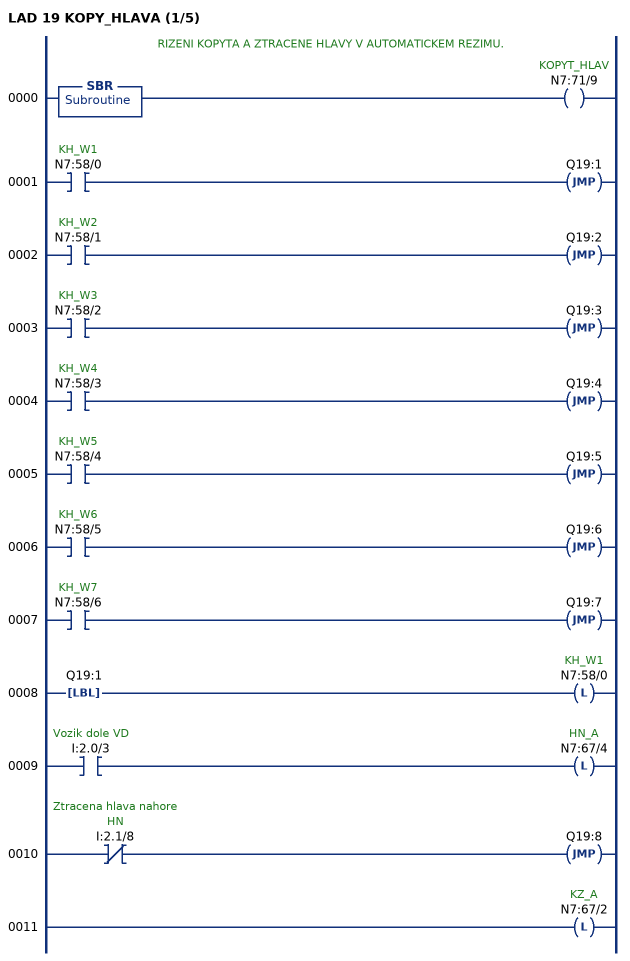
% Rung: 0 %
% RIZENI KOPYTA A ZTRACENE HLAVY V AUTOMATICKEM REZIMU. %
SOR SBR OTE N7:71/9 EOR
%   N7:71/9  KOPYT_HLAV %
% Rung: 1 %
SOR XIC N7:58/0 JMP Q19:1 EOR
%   N7:58/0  KH_W1 %
% Rung: 2 %
SOR XIC N7:58/1 JMP Q19:2 EOR
%   N7:58/1  KH_W2 %
% Rung: 3 %
SOR XIC N7:58/2 JMP Q19:3 EOR
%   N7:58/2  KH_W3 %
% Rung: 4 %
SOR XIC N7:58/3 JMP Q19:4 EOR
%   N7:58/3  KH_W4 %
% Rung: 5 %
SOR XIC N7:58/4 JMP Q19:5 EOR
%   N7:58/4  KH_W5 %
% Rung: 6 %
SOR XIC N7:58/5 JMP Q19:6 EOR
%   N7:58/5  KH_W6 %
% Rung: 7 %
SOR XIC N7:58/6 JMP Q19:7 EOR
%   N7:58/6  KH_W7 %
% Rung: 8 %
SOR LBL Q19:1 OTL N7:58/0 EOR
%   N7:58/0  KH_W1 %
% Rung: 9 %
SOR XIC I:2.0/3 OTL N7:67/4 EOR
%   I:2.0/3  VD  "Vozik dole" %
%   N7:67/4  HN_A %
% Rung: 10 %
SOR XIO I:2.1/8 JMP Q19:8 EOR
%   I:2.1/8  HN  "Ztracena hlava nahore" %
% Rung: 11 %
SOR OTL N7:67/2 EOR
%   N7:67/2  KZ_A %

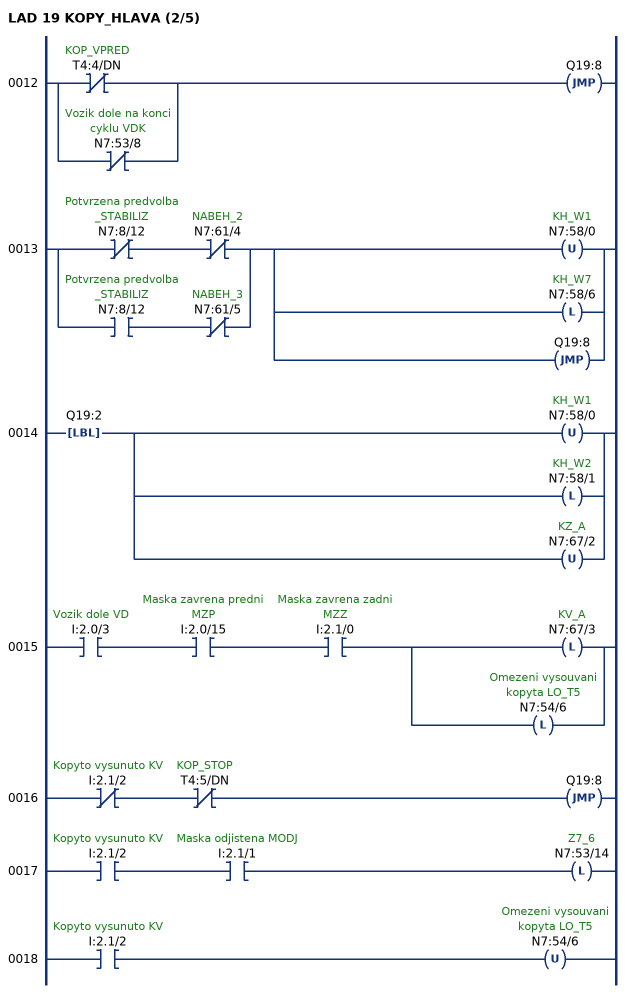
% Rung: 12 %
SOR BST XIO T4:4/DN NXB XIO N7:53/8 BND JMP Q19:8 EOR
%   T4:4/DN  KOP_VPRED %
%   N7:53/8  VDK  "Vozik dole na konci cyklu" %
% Rung: 13 %
SOR BST XIO N7:8/12 XIO N7:61/4 NXB XIC N7:8/12 XIO N7:61/5 BND BST OTU N7:58/0 NXB OTL N7:58/6 NXB JMP Q19:8 BND EOR
%   N7:8/12  _STABILIZ  "Potvrzena predvolba" %
%   N7:61/4  NABEH_2 %
%   N7:61/5  NABEH_3 %
%   N7:58/0  KH_W1 %
%   N7:58/6  KH_W7 %
% Rung: 14 %
SOR LBL Q19:2 BST OTU N7:58/0 NXB OTL N7:58/1 NXB OTU N7:67/2 BND EOR
%   N7:58/0  KH_W1 %
%   N7:58/1  KH_W2 %
%   N7:67/2  KZ_A %
% Rung: 15 %
SOR XIC I:2.0/3 XIC I:2.0/15 XIC I:2.1/0 BST OTL N7:67/3 NXB OTL N7:54/6 BND EOR
%   I:2.0/3  VD  "Vozik dole" %
%   I:2.0/15  MZP  "Maska zavrena predni" %
%   I:2.1/0  MZZ  "Maska zavrena zadni" %
%   N7:67/3  KV_A %
%   N7:54/6  LO_T5  "Omezeni vysouvani kopyta" %
% Rung: 16 %
SOR XIO I:2.1/2 XIO T4:5/DN JMP Q19:8 EOR
%   I:2.1/2  KV  "Kopyto vysunuto" %
%   T4:5/DN  KOP_STOP %
% Rung: 17 %
SOR XIC I:2.1/2 XIC I:2.1/1 OTL N7:53/14 EOR
%   I:2.1/2  KV  "Kopyto vysunuto" %
%   I:2.1/1  MODJ  "Maska odjistena" %
%   N7:53/14  Z7_6 %
% Rung: 18 %
SOR XIC I:2.1/2 OTU N7:54/6 EOR
%   I:2.1/2  KV  "Kopyto vysunuto" %
%   N7:54/6  LO_T5  "Omezeni vysouvani kopyta" %

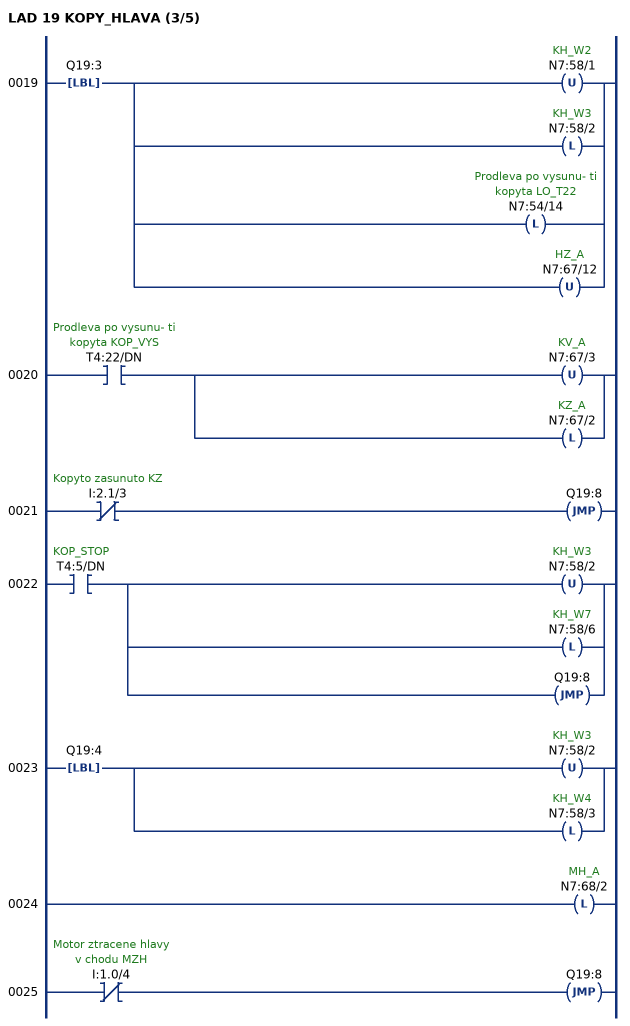
% Rung: 19 %
SOR LBL Q19:3 BST OTU N7:58/1 NXB OTL N7:58/2 NXB OTL N7:54/14 NXB OTU N7:67/12 BND EOR
%   N7:58/1  KH_W2 %
%   N7:58/2  KH_W3 %
%   N7:54/14  LO_T22  "Prodleva po vysunu- ti kopyta" %
%   N7:67/12  HZ_A %
% Rung: 20 %
SOR XIC T4:22/DN BST OTU N7:67/3 NXB OTL N7:67/2 BND EOR
%   T4:22/DN  KOP_VYS  "Prodleva po vysunu- ti kopyta" %
%   N7:67/3  KV_A %
%   N7:67/2  KZ_A %
% Rung: 21 %
SOR XIO I:2.1/3 JMP Q19:8 EOR
%   I:2.1/3  KZ  "Kopyto zasunuto" %
% Rung: 22 %
SOR XIC T4:5/DN BST OTU N7:58/2 NXB OTL N7:58/6 NXB JMP Q19:8 BND EOR
%   T4:5/DN  KOP_STOP %
%   N7:58/2  KH_W3 %
%   N7:58/6  KH_W7 %
% Rung: 23 %
SOR LBL Q19:4 BST OTU N7:58/2 NXB OTL N7:58/3 BND EOR
%   N7:58/2  KH_W3 %
%   N7:58/3  KH_W4 %
% Rung: 24 %
SOR OTL N7:68/2 EOR
%   N7:68/2  MH_A %
% Rung: 25 %
SOR XIO I:1.0/4 JMP Q19:8 EOR
%   I:1.0/4  MZH  "Motor ztracene hlavy v chodu" %

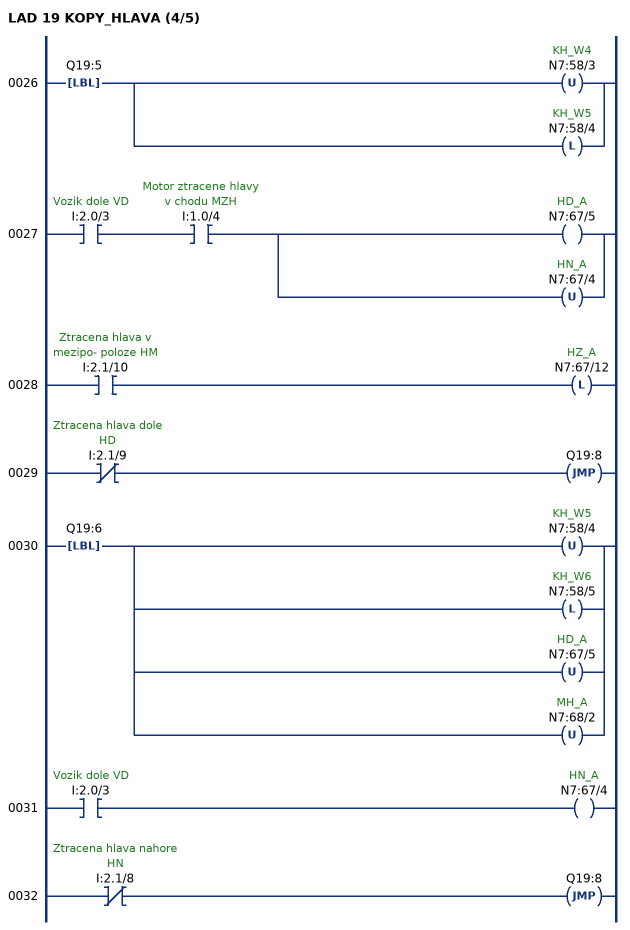
% Rung: 26 %
SOR LBL Q19:5 BST OTU N7:58/3 NXB OTL N7:58/4 BND EOR
%   N7:58/3  KH_W4 %
%   N7:58/4  KH_W5 %
% Rung: 27 %
SOR XIC I:2.0/3 XIC I:1.0/4 BST OTE N7:67/5 NXB OTU N7:67/4 BND EOR
%   I:2.0/3  VD  "Vozik dole" %
%   I:1.0/4  MZH  "Motor ztracene hlavy v chodu" %
%   N7:67/5  HD_A %
%   N7:67/4  HN_A %
% Rung: 28 %
SOR XIC I:2.1/10 OTL N7:67/12 EOR
%   I:2.1/10  HM  "Ztracena hlava v mezipo- poloze" %
%   N7:67/12  HZ_A %
% Rung: 29 %
SOR XIO I:2.1/9 JMP Q19:8 EOR
%   I:2.1/9  HD  "Ztracena hlava dole" %
% Rung: 30 %
SOR LBL Q19:6 BST OTU N7:58/4 NXB OTL N7:58/5 NXB OTU N7:67/5 NXB OTU N7:68/2 BND EOR
%   N7:58/4  KH_W5 %
%   N7:58/5  KH_W6 %
%   N7:67/5  HD_A %
%   N7:68/2  MH_A %
% Rung: 31 %
SOR XIC I:2.0/3 OTE N7:67/4 EOR
%   I:2.0/3  VD  "Vozik dole" %
%   N7:67/4  HN_A %
% Rung: 32 %
SOR XIO I:2.1/8 JMP Q19:8 EOR
%   I:2.1/8  HN  "Ztracena hlava nahore" %

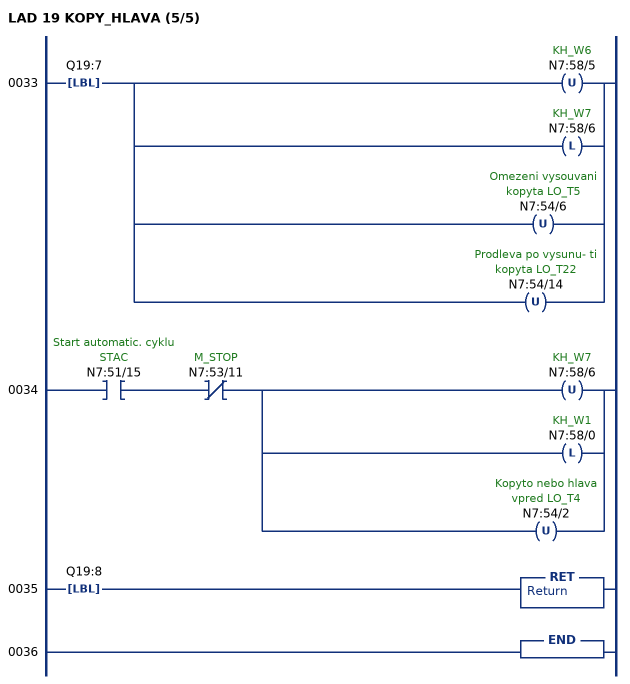
% Rung: 33 %
SOR LBL Q19:7 BST OTU N7:58/5 NXB OTL N7:58/6 NXB OTU N7:54/6 NXB OTU N7:54/14 BND EOR
%   N7:58/5  KH_W6 %
%   N7:58/6  KH_W7 %
%   N7:54/6  LO_T5  "Omezeni vysouvani kopyta" %
%   N7:54/14  LO_T22  "Prodleva po vysunu- ti kopyta" %
% Rung: 34 %
SOR XIC N7:51/15 XIO N7:53/11 BST OTU N7:58/6 NXB OTL N7:58/0 NXB OTU N7:54/2 BND EOR
%   N7:51/15  STAC  "Start automatic. cyklu" %
%   N7:53/11  M_STOP %
%   N7:58/6  KH_W7 %
%   N7:58/0  KH_W1 %
%   N7:54/2  LO_T4  "Kopyto nebo hlava vpred" %
% Rung: 35 %
SOR LBL Q19:8 RET EOR
% Rung: 36 %
SOR END EOR

LADDER 20 "STABILIZ"
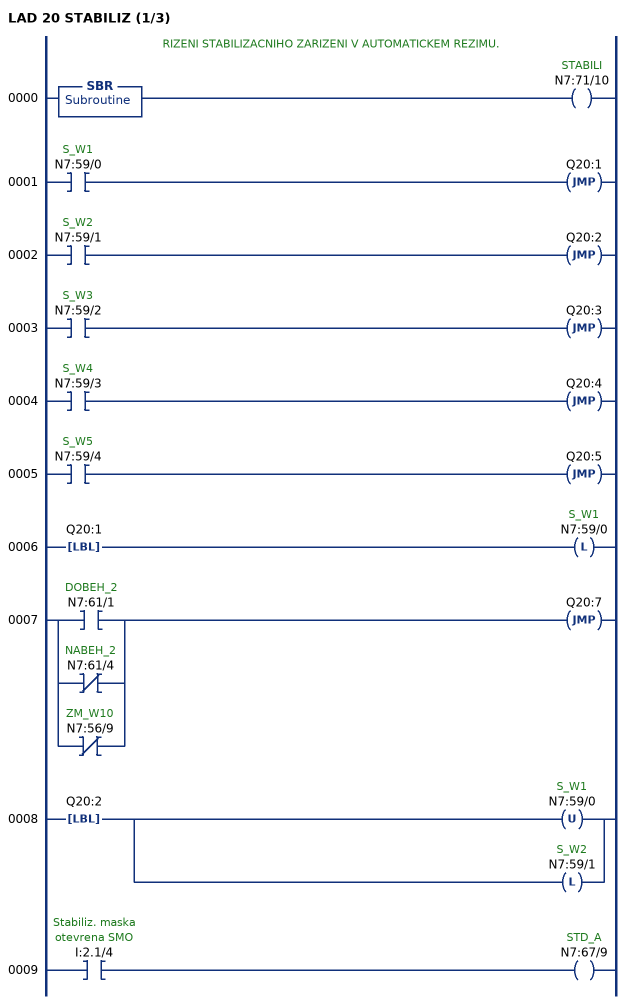
% Rung: 0 %
% RIZENI STABILIZACNIHO ZARIZENI V AUTOMATICKEM REZIMU. %
SOR SBR OTE N7:71/10 EOR
%   N7:71/10  STABILI %
% Rung: 1 %
SOR XIC N7:59/0 JMP Q20:1 EOR
%   N7:59/0  S_W1 %
% Rung: 2 %
SOR XIC N7:59/1 JMP Q20:2 EOR
%   N7:59/1  S_W2 %
% Rung: 3 %
SOR XIC N7:59/2 JMP Q20:3 EOR
%   N7:59/2  S_W3 %
% Rung: 4 %
SOR XIC N7:59/3 JMP Q20:4 EOR
%   N7:59/3  S_W4 %
% Rung: 5 %
SOR XIC N7:59/4 JMP Q20:5 EOR
%   N7:59/4  S_W5 %
% Rung: 6 %
SOR LBL Q20:1 OTL N7:59/0 EOR
%   N7:59/0  S_W1 %
% Rung: 7 %
SOR BST XIC N7:61/1 NXB XIO N7:61/4 NXB XIO N7:56/9 BND JMP Q20:7 EOR
%   N7:61/1  DOBEH_2 %
%   N7:61/4  NABEH_2 %
%   N7:56/9  ZM_W10 %
% Rung: 8 %
SOR LBL Q20:2 BST OTU N7:59/0 NXB OTL N7:59/1 BND EOR
%   N7:59/0  S_W1 %
%   N7:59/1  S_W2 %
% Rung: 9 %
SOR XIC I:2.1/4 OTE N7:67/9 EOR
%   I:2.1/4  SMO  "Stabiliz. maska otevrena" %
%   N7:67/9  STD_A %

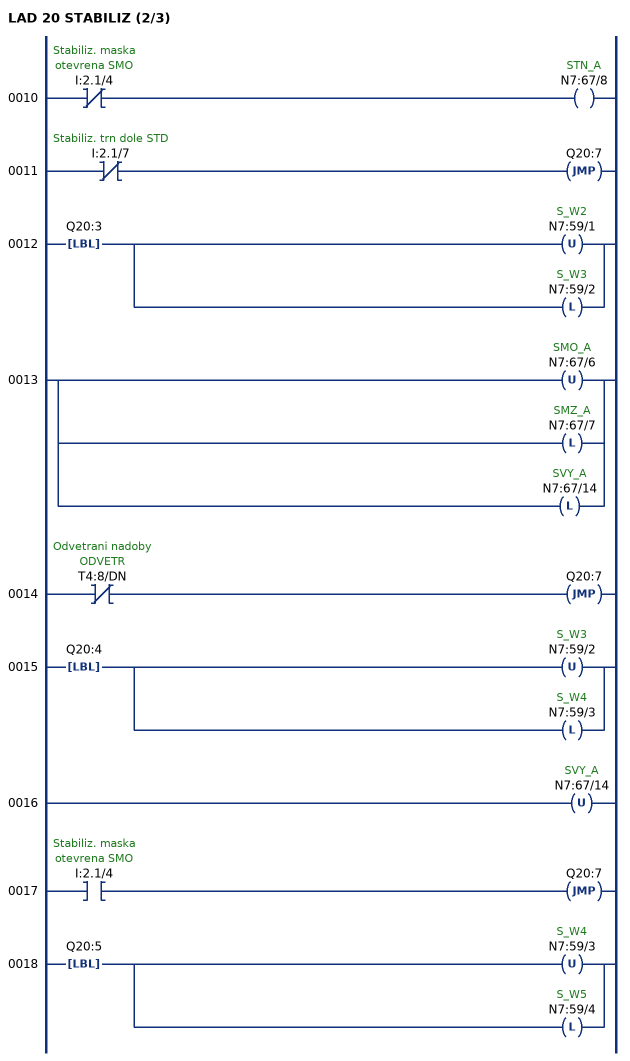
% Rung: 10 %
SOR XIO I:2.1/4 OTE N7:67/8 EOR
%   I:2.1/4  SMO  "Stabiliz. maska otevrena" %
%   N7:67/8  STN_A %
% Rung: 11 %
SOR XIO I:2.1/7 JMP Q20:7 EOR
%   I:2.1/7  STD  "Stabiliz. trn dole" %
% Rung: 12 %
SOR LBL Q20:3 BST OTU N7:59/1 NXB OTL N7:59/2 BND EOR
%   N7:59/1  S_W2 %
%   N7:59/2  S_W3 %
% Rung: 13 %
SOR BST OTU N7:67/6 NXB OTL N7:67/7 NXB OTL N7:67/14 BND EOR
%   N7:67/6  SMO_A %
%   N7:67/7  SMZ_A %
%   N7:67/14  SVY_A %
% Rung: 14 %
SOR XIO T4:8/DN JMP Q20:7 EOR
%   T4:8/DN  ODVETR  "Odvetrani nadoby" %
% Rung: 15 %
SOR LBL Q20:4 BST OTU N7:59/2 NXB OTL N7:59/3 BND EOR
%   N7:59/2  S_W3 %
%   N7:59/3  S_W4 %
% Rung: 16 %
SOR OTU N7:67/14 EOR
%   N7:67/14  SVY_A %
% Rung: 17 %
SOR XIC I:2.1/4 JMP Q20:7 EOR
%   I:2.1/4  SMO  "Stabiliz. maska otevrena" %
% Rung: 18 %
SOR LBL Q20:5 BST OTU N7:59/3 NXB OTL N7:59/4 BND EOR
%   N7:59/3  S_W4 %
%   N7:59/4  S_W5 %

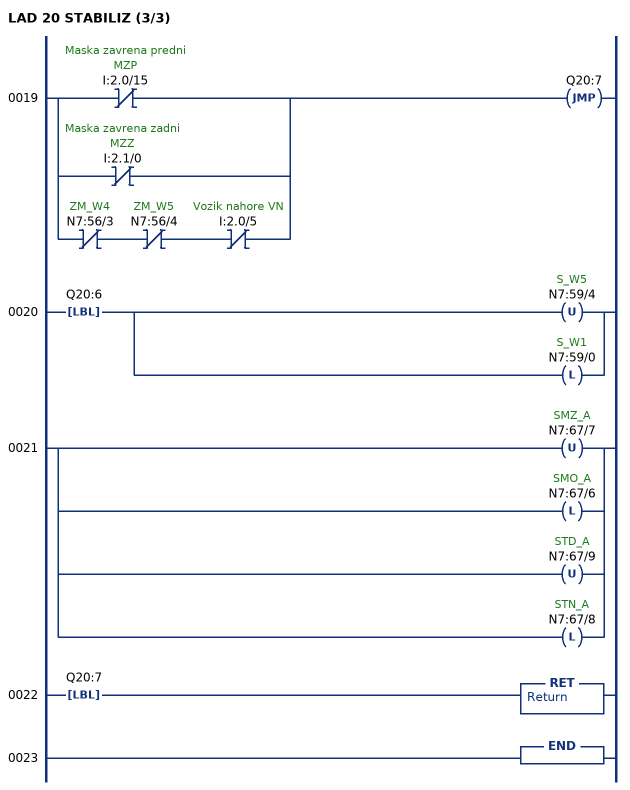
% Rung: 19 %
SOR BST XIO I:2.0/15 NXB XIO I:2.1/0 NXB XIO N7:56/3 XIO N7:56/4 XIO I:2.0/5 BND JMP Q20:7 EOR
%   I:2.0/15  MZP  "Maska zavrena predni" %
%   I:2.1/0  MZZ  "Maska zavrena zadni" %
%   N7:56/3  ZM_W4 %
%   N7:56/4  ZM_W5 %
%   I:2.0/5  VN  "Vozik nahore" %
% Rung: 20 %
SOR LBL Q20:6 BST OTU N7:59/4 NXB OTL N7:59/0 BND EOR
%   N7:59/4  S_W5 %
%   N7:59/0  S_W1 %
% Rung: 21 %
SOR BST OTU N7:67/7 NXB OTL N7:67/6 NXB OTU N7:67/9 NXB OTL N7:67/8 BND EOR
%   N7:67/7  SMZ_A %
%   N7:67/6  SMO_A %
%   N7:67/9  STD_A %
%   N7:67/8  STN_A %
% Rung: 22 %
SOR LBL Q20:7 RET EOR
% Rung: 23 %
SOR END EOR

LADDER 21 "ODDEL_IMP"
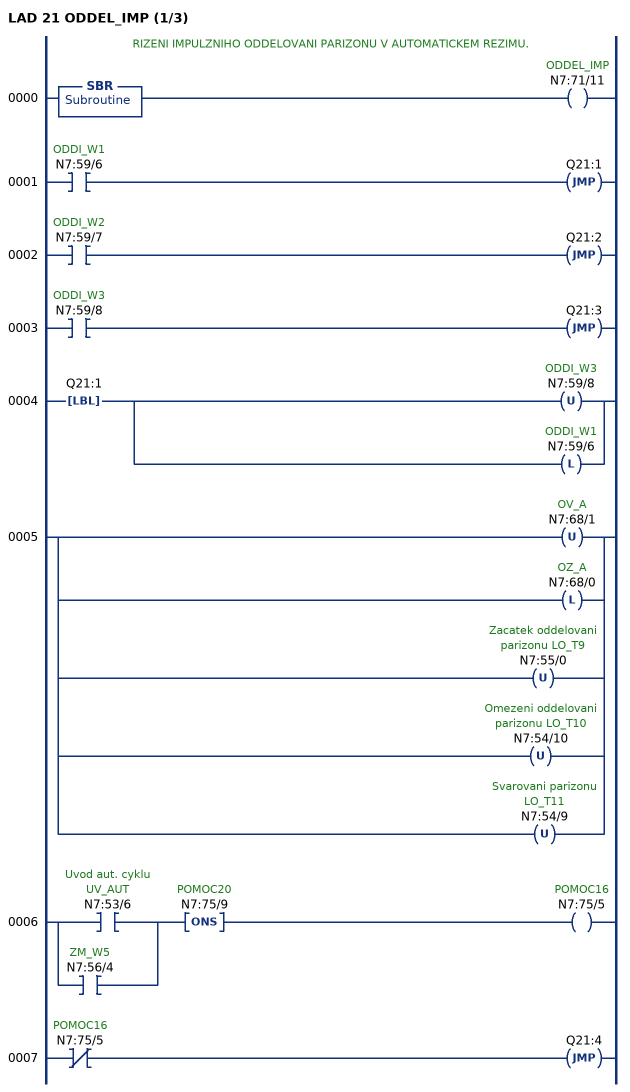
% Rung: 0 %
% RIZENI IMPULZNIHO ODDELOVANI PARIZONU V AUTOMATICKEM REZIMU. %
SOR SBR OTE N7:71/11 EOR
%   N7:71/11  ODDEL_IMP %
% Rung: 1 %
SOR XIC N7:59/6 JMP Q21:1 EOR
%   N7:59/6  ODDI_W1 %
% Rung: 2 %
SOR XIC N7:59/7 JMP Q21:2 EOR
%   N7:59/7  ODDI_W2 %
% Rung: 3 %
SOR XIC N7:59/8 JMP Q21:3 EOR
%   N7:59/8  ODDI_W3 %
% Rung: 4 %
SOR LBL Q21:1 BST OTU N7:59/8 NXB OTL N7:59/6 BND EOR
%   N7:59/8  ODDI_W3 %
%   N7:59/6  ODDI_W1 %
% Rung: 5 %
SOR BST OTU N7:68/1 NXB OTL N7:68/0 NXB OTU N7:55/0 NXB OTU N7:54/10 NXB OTU N7:54/9 BND EOR
%   N7:68/1  OV_A %
%   N7:68/0  OZ_A %
%   N7:55/0  LO_T9  "Zacatek oddelovani parizonu" %
%   N7:54/10  LO_T10  "Omezeni oddelovani parizonu" %
%   N7:54/9  LO_T11  "Svarovani parizonu" %
% Rung: 6 %
SOR BST XIC N7:53/6 NXB XIC N7:56/4 BND OSR N7:75/9 OTE N7:75/5 EOR
%   N7:53/6  UV_AUT  "Uvod aut. cyklu" %
%   N7:56/4  ZM_W5 %
%   N7:75/9  POMOC20 %
%   N7:75/5  POMOC16 %
% Rung: 7 %
SOR XIO N7:75/5 JMP Q21:4 EOR
%   N7:75/5  POMOC16 %

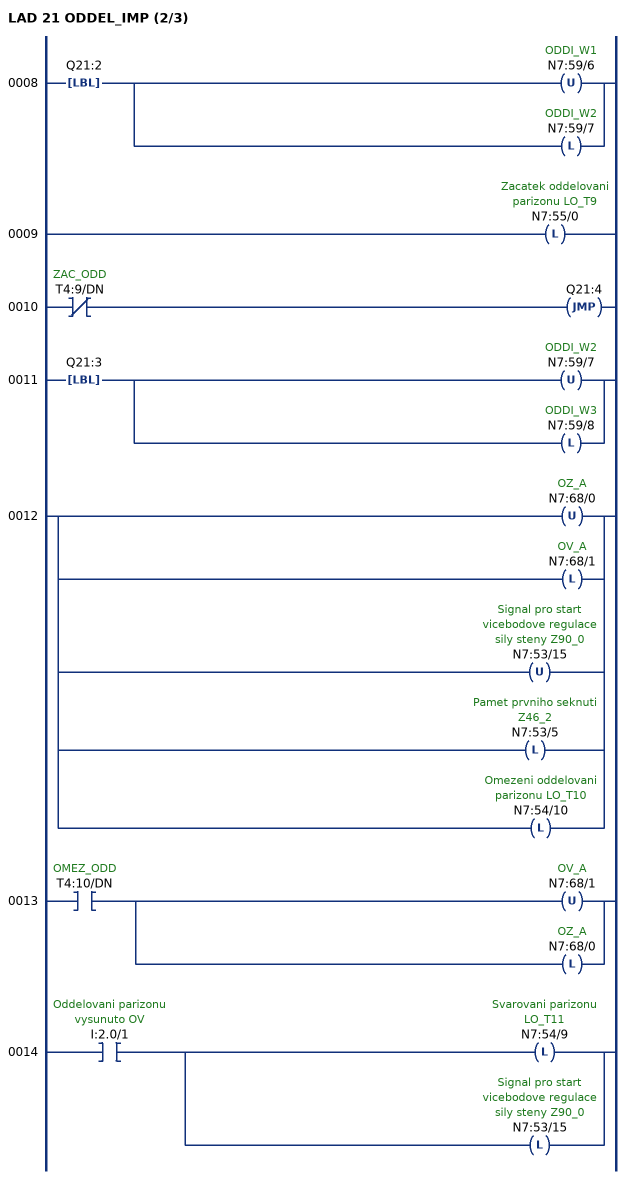
% Rung: 8 %
SOR LBL Q21:2 BST OTU N7:59/6 NXB OTL N7:59/7 BND EOR
%   N7:59/6  ODDI_W1 %
%   N7:59/7  ODDI_W2 %
% Rung: 9 %
SOR OTL N7:55/0 EOR
%   N7:55/0  LO_T9  "Zacatek oddelovani parizonu" %
% Rung: 10 %
SOR XIO T4:9/DN JMP Q21:4 EOR
%   T4:9/DN  ZAC_ODD %
% Rung: 11 %
SOR LBL Q21:3 BST OTU N7:59/7 NXB OTL N7:59/8 BND EOR
%   N7:59/7  ODDI_W2 %
%   N7:59/8  ODDI_W3 %
% Rung: 12 %
SOR BST OTU N7:68/0 NXB OTL N7:68/1 NXB OTU N7:53/15 NXB OTL N7:53/5 NXB OTL N7:54/10 BND EOR
%   N7:68/0  OZ_A %
%   N7:68/1  OV_A %
%   N7:53/15  Z90_0  "Signal pro start vicebodove regulace sily steny" %
%   N7:53/5  Z46_2  "Pamet prvniho seknuti" %
%   N7:54/10  LO_T10  "Omezeni oddelovani parizonu" %
% Rung: 13 %
SOR XIC T4:10/DN BST OTU N7:68/1 NXB OTL N7:68/0 BND EOR
%   T4:10/DN  OMEZ_ODD %
%   N7:68/1  OV_A %
%   N7:68/0  OZ_A %
% Rung: 14 %
SOR XIC I:2.0/1 BST OTL N7:54/9 NXB OTL N7:53/15 BND EOR
%   I:2.0/1  OV  "Oddelovani parizonu vysunuto" %
%   N7:54/9  LO_T11  "Svarovani parizonu" %
%   N7:53/15  Z90_0  "Signal pro start vicebodove regulace sily steny" %

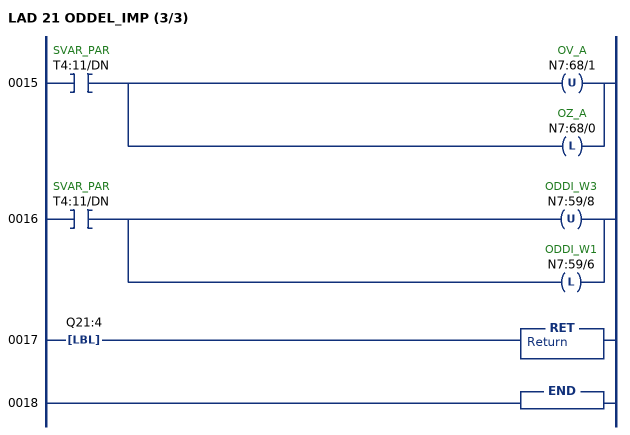
% Rung: 15 %
SOR XIC T4:11/DN BST OTU N7:68/1 NXB OTL N7:68/0 BND EOR
%   T4:11/DN  SVAR_PAR %
%   N7:68/1  OV_A %
%   N7:68/0  OZ_A %
% Rung: 16 %
SOR XIC T4:11/DN BST OTU N7:59/8 NXB OTL N7:59/6 BND EOR
%   T4:11/DN  SVAR_PAR %
%   N7:59/8  ODDI_W3 %
%   N7:59/6  ODDI_W1 %
% Rung: 17 %
SOR LBL Q21:4 RET EOR
% Rung: 18 %
SOR END EOR

LADDER 22 "ODDEL_RS"
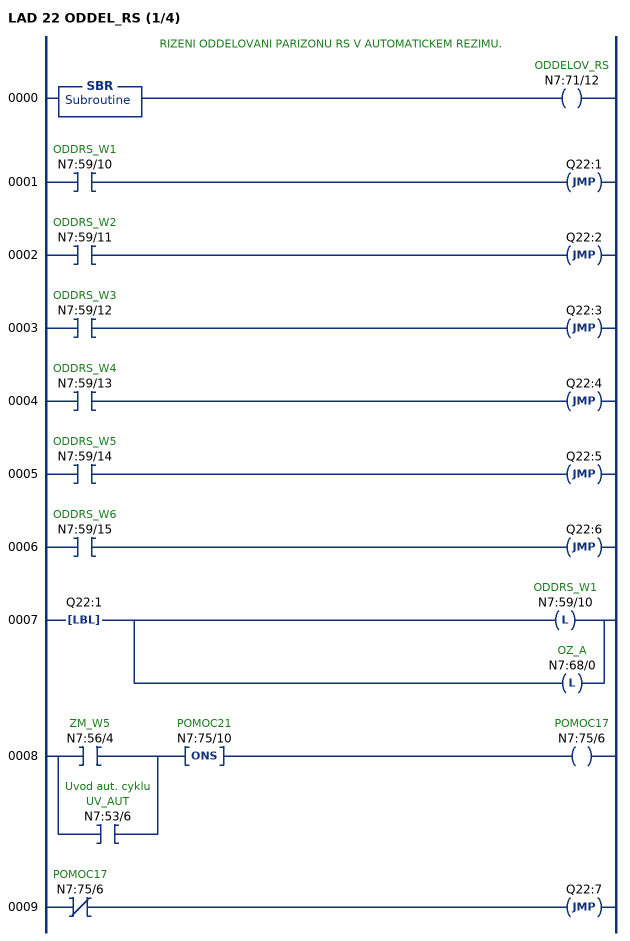
% Rung: 0 %
% RIZENI ODDELOVANI PARIZONU RS V AUTOMATICKEM REZIMU. %
SOR SBR OTE N7:71/12 EOR
%   N7:71/12  ODDELOV_RS %
% Rung: 1 %
SOR XIC N7:59/10 JMP Q22:1 EOR
%   N7:59/10  ODDRS_W1 %
% Rung: 2 %
SOR XIC N7:59/11 JMP Q22:2 EOR
%   N7:59/11  ODDRS_W2 %
% Rung: 3 %
SOR XIC N7:59/12 JMP Q22:3 EOR
%   N7:59/12  ODDRS_W3 %
% Rung: 4 %
SOR XIC N7:59/13 JMP Q22:4 EOR
%   N7:59/13  ODDRS_W4 %
% Rung: 5 %
SOR XIC N7:59/14 JMP Q22:5 EOR
%   N7:59/14  ODDRS_W5 %
% Rung: 6 %
SOR XIC N7:59/15 JMP Q22:6 EOR
%   N7:59/15  ODDRS_W6 %
% Rung: 7 %
SOR LBL Q22:1 BST OTL N7:59/10 NXB OTL N7:68/0 BND EOR
%   N7:59/10  ODDRS_W1 %
%   N7:68/0  OZ_A %
% Rung: 8 %
SOR BST XIC N7:56/4 NXB XIC N7:53/6 BND OSR N7:75/10 OTE N7:75/6 EOR
%   N7:56/4  ZM_W5 %
%   N7:53/6  UV_AUT  "Uvod aut. cyklu" %
%   N7:75/10  POMOC21 %
%   N7:75/6  POMOC17 %
% Rung: 9 %
SOR XIO N7:75/6 JMP Q22:7 EOR
%   N7:75/6  POMOC17 %

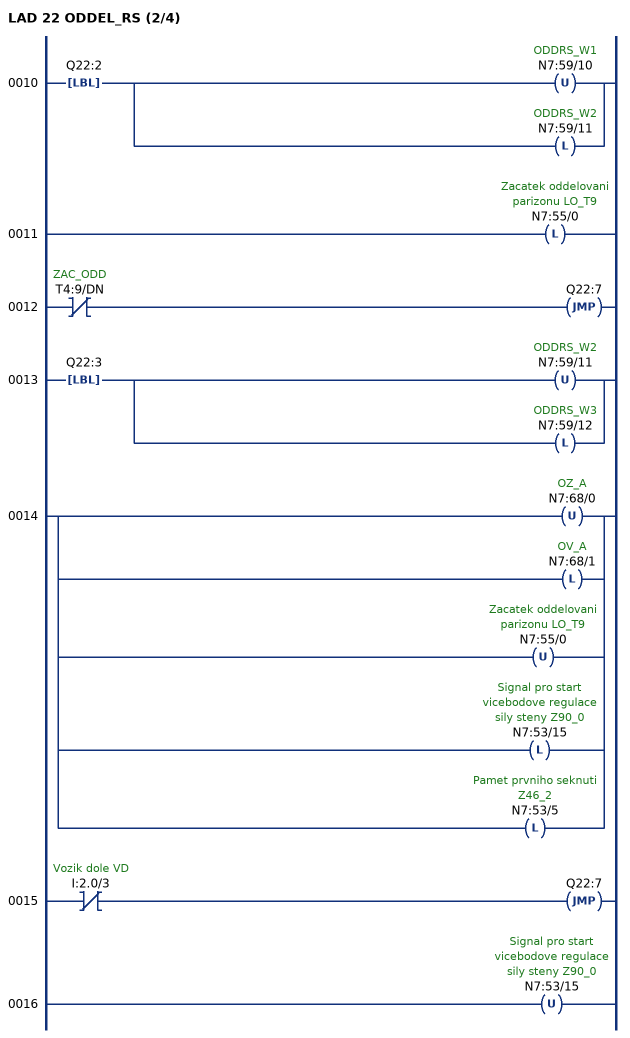
% Rung: 10 %
SOR LBL Q22:2 BST OTU N7:59/10 NXB OTL N7:59/11 BND EOR
%   N7:59/10  ODDRS_W1 %
%   N7:59/11  ODDRS_W2 %
% Rung: 11 %
SOR OTL N7:55/0 EOR
%   N7:55/0  LO_T9  "Zacatek oddelovani parizonu" %
% Rung: 12 %
SOR XIO T4:9/DN JMP Q22:7 EOR
%   T4:9/DN  ZAC_ODD %
% Rung: 13 %
SOR LBL Q22:3 BST OTU N7:59/11 NXB OTL N7:59/12 BND EOR
%   N7:59/11  ODDRS_W2 %
%   N7:59/12  ODDRS_W3 %
% Rung: 14 %
SOR BST OTU N7:68/0 NXB OTL N7:68/1 NXB OTU N7:55/0 NXB OTL N7:53/15 NXB OTL N7:53/5 BND EOR
%   N7:68/0  OZ_A %
%   N7:68/1  OV_A %
%   N7:55/0  LO_T9  "Zacatek oddelovani parizonu" %
%   N7:53/15  Z90_0  "Signal pro start vicebodove regulace sily steny" %
%   N7:53/5  Z46_2  "Pamet prvniho seknuti" %
% Rung: 15 %
SOR XIO I:2.0/3 JMP Q22:7 EOR
%   I:2.0/3  VD  "Vozik dole" %
% Rung: 16 %
SOR OTU N7:53/15 EOR
%   N7:53/15  Z90_0  "Signal pro start vicebodove regulace sily steny" %

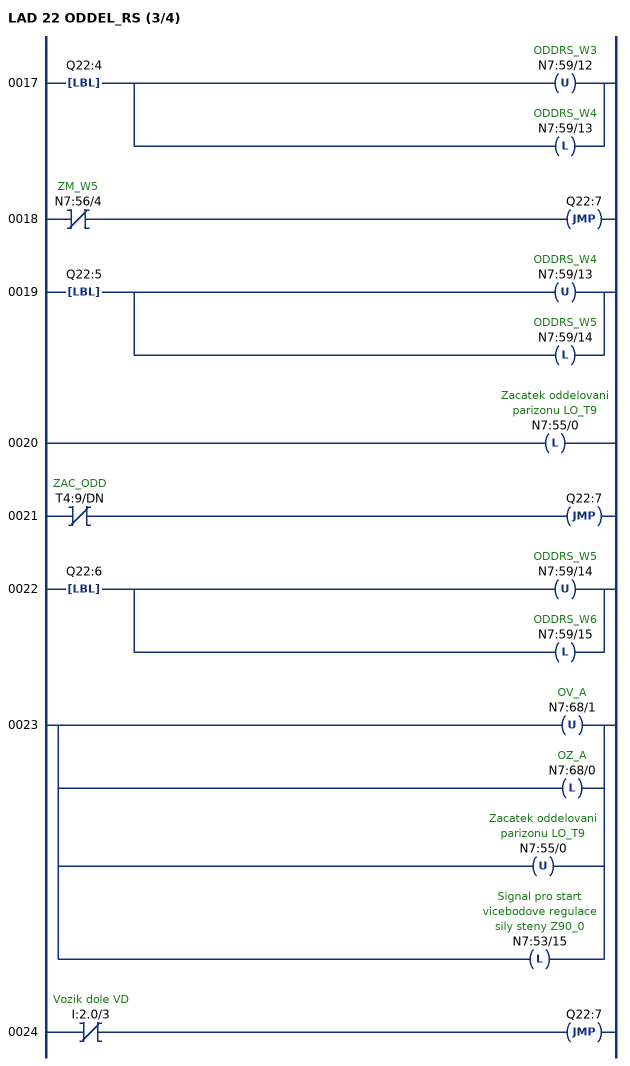
% Rung: 17 %
SOR LBL Q22:4 BST OTU N7:59/12 NXB OTL N7:59/13 BND EOR
%   N7:59/12  ODDRS_W3 %
%   N7:59/13  ODDRS_W4 %
% Rung: 18 %
SOR XIO N7:56/4 JMP Q22:7 EOR
%   N7:56/4  ZM_W5 %
% Rung: 19 %
SOR LBL Q22:5 BST OTU N7:59/13 NXB OTL N7:59/14 BND EOR
%   N7:59/13  ODDRS_W4 %
%   N7:59/14  ODDRS_W5 %
% Rung: 20 %
SOR OTL N7:55/0 EOR
%   N7:55/0  LO_T9  "Zacatek oddelovani parizonu" %
% Rung: 21 %
SOR XIO T4:9/DN JMP Q22:7 EOR
%   T4:9/DN  ZAC_ODD %
% Rung: 22 %
SOR LBL Q22:6 BST OTU N7:59/14 NXB OTL N7:59/15 BND EOR
%   N7:59/14  ODDRS_W5 %
%   N7:59/15  ODDRS_W6 %
% Rung: 23 %
SOR BST OTU N7:68/1 NXB OTL N7:68/0 NXB OTU N7:55/0 NXB OTL N7:53/15 BND EOR
%   N7:68/1  OV_A %
%   N7:68/0  OZ_A %
%   N7:55/0  LO_T9  "Zacatek oddelovani parizonu" %
%   N7:53/15  Z90_0  "Signal pro start vicebodove regulace sily steny" %
% Rung: 24 %
SOR XIO I:2.0/3 JMP Q22:7 EOR
%   I:2.0/3  VD  "Vozik dole" %

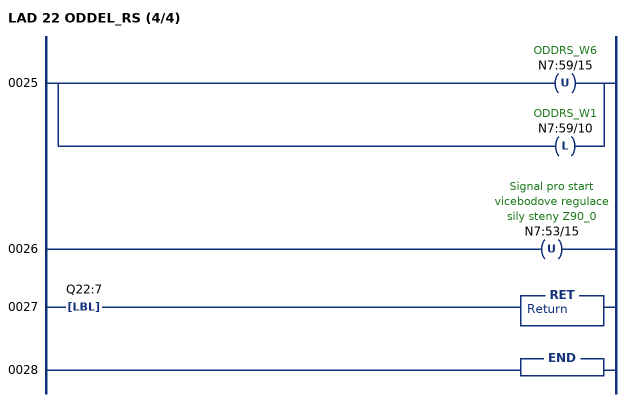
% Rung: 25 %
SOR BST OTU N7:59/15 NXB OTL N7:59/10 BND EOR
%   N7:59/15  ODDRS_W6 %
%   N7:59/10  ODDRS_W1 %
% Rung: 26 %
SOR OTU N7:53/15 EOR
%   N7:53/15  Z90_0  "Signal pro start vicebodove regulace sily steny" %
% Rung: 27 %
SOR LBL Q22:7 RET EOR
% Rung: 28 %
SOR END EOR

LADDER 23 "PODPUR_VZD"
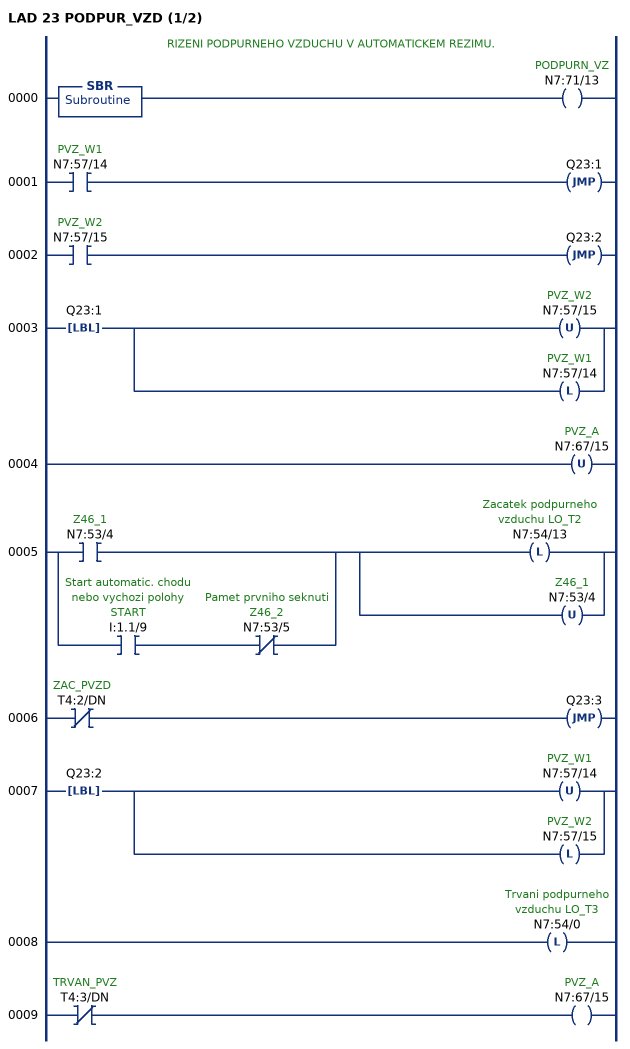
% Rung: 0 %
% RIZENI PODPURNEHO VZDUCHU V AUTOMATICKEM REZIMU. %
SOR SBR OTE N7:71/13 EOR
%   N7:71/13  PODPURN_VZ %
% Rung: 1 %
SOR XIC N7:57/14 JMP Q23:1 EOR
%   N7:57/14  PVZ_W1 %
% Rung: 2 %
SOR XIC N7:57/15 JMP Q23:2 EOR
%   N7:57/15  PVZ_W2 %
% Rung: 3 %
SOR LBL Q23:1 BST OTU N7:57/15 NXB OTL N7:57/14 BND EOR
%   N7:57/15  PVZ_W2 %
%   N7:57/14  PVZ_W1 %
% Rung: 4 %
SOR OTU N7:67/15 EOR
%   N7:67/15  PVZ_A %
% Rung: 5 %
SOR BST XIC N7:53/4 NXB XIC I:1.1/9 XIO N7:53/5 BND BST OTL N7:54/13 NXB OTU N7:53/4 BND EOR
%   N7:53/4  Z46_1 %
%   I:1.1/9  START  "Start automatic. chodu nebo vychozi polohy" %
%   N7:53/5  Z46_2  "Pamet prvniho seknuti" %
%   N7:54/13  LO_T2  "Zacatek podpurneho vzduchu" %
% Rung: 6 %
SOR XIO T4:2/DN JMP Q23:3 EOR
%   T4:2/DN  ZAC_PVZD %
% Rung: 7 %
SOR LBL Q23:2 BST OTU N7:57/14 NXB OTL N7:57/15 BND EOR
%   N7:57/14  PVZ_W1 %
%   N7:57/15  PVZ_W2 %
% Rung: 8 %
SOR OTL N7:54/0 EOR
%   N7:54/0  LO_T3  "Trvani podpurneho vzduchu" %
% Rung: 9 %
SOR XIO T4:3/DN OTE N7:67/15 EOR
%   T4:3/DN  TRVAN_PVZ %
%   N7:67/15  PVZ_A %

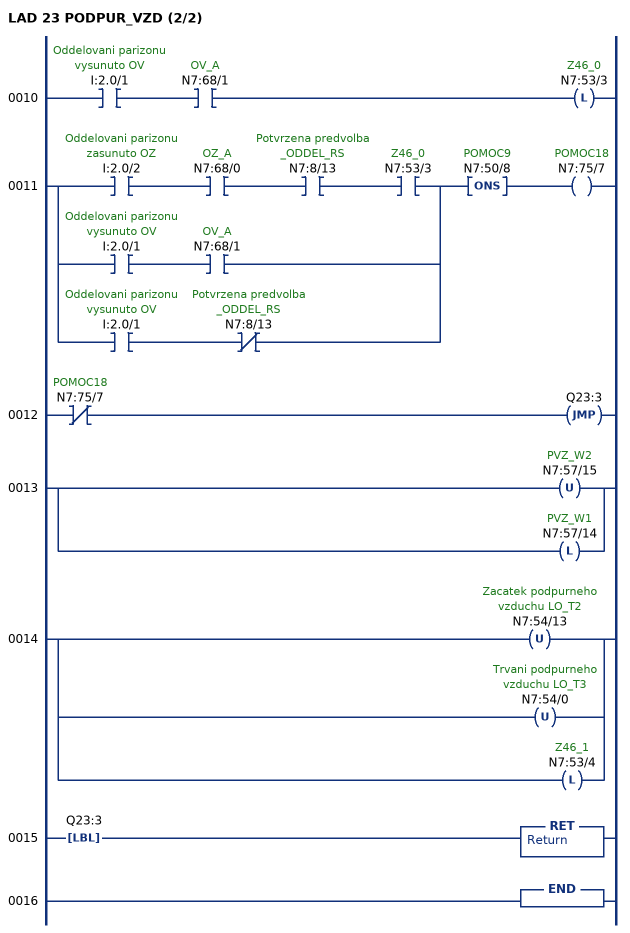
% Rung: 10 %
SOR XIC I:2.0/1 XIC N7:68/1 OTL N7:53/3 EOR
%   I:2.0/1  OV  "Oddelovani parizonu vysunuto" %
%   N7:68/1  OV_A %
%   N7:53/3  Z46_0 %
% Rung: 11 %
SOR BST XIC I:2.0/2 XIC N7:68/0 XIC N7:8/13 XIC N7:53/3 NXB XIC I:2.0/1 XIC N7:68/1 NXB XIC I:2.0/1 XIO N7:8/13 BND OSR N7:50/8 OTE N7:75/7 EOR
%   I:2.0/2  OZ  "Oddelovani parizonu zasunuto" %
%   N7:68/0  OZ_A %
%   N7:8/13  _ODDEL_RS  "Potvrzena predvolba" %
%   N7:53/3  Z46_0 %
%   I:2.0/1  OV  "Oddelovani parizonu vysunuto" %
%   N7:68/1  OV_A %
%   N7:50/8  POMOC9 %
%   N7:75/7  POMOC18 %
% Rung: 12 %
SOR XIO N7:75/7 JMP Q23:3 EOR
%   N7:75/7  POMOC18 %
% Rung: 13 %
SOR BST OTU N7:57/15 NXB OTL N7:57/14 BND EOR
%   N7:57/15  PVZ_W2 %
%   N7:57/14  PVZ_W1 %
% Rung: 14 %
SOR BST OTU N7:54/13 NXB OTU N7:54/0 NXB OTL N7:53/4 BND EOR
%   N7:54/13  LO_T2  "Zacatek podpurneho vzduchu" %
%   N7:54/0  LO_T3  "Trvani podpurneho vzduchu" %
%   N7:53/4  Z46_1 %
% Rung: 15 %
SOR LBL Q23:3 RET EOR
% Rung: 16 %
SOR END EOR

LADDER 24 "VYFUK_TRN"
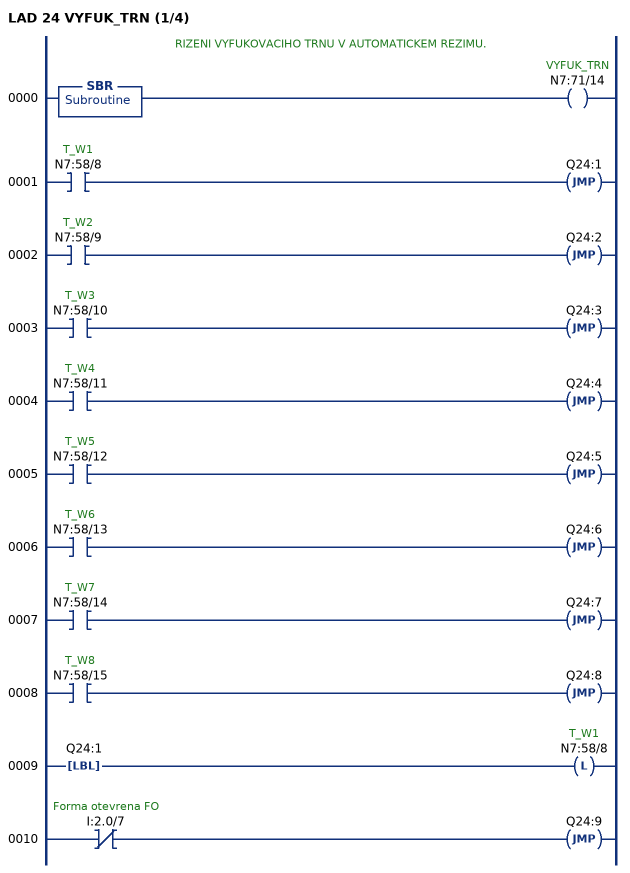
% Rung: 0 %
% RIZENI VYFUKOVACIHO TRNU V AUTOMATICKEM REZIMU. %
SOR SBR OTE N7:71/14 EOR
%   N7:71/14  VYFUK_TRN %
% Rung: 1 %
SOR XIC N7:58/8 JMP Q24:1 EOR
%   N7:58/8  T_W1 %
% Rung: 2 %
SOR XIC N7:58/9 JMP Q24:2 EOR
%   N7:58/9  T_W2 %
% Rung: 3 %
SOR XIC N7:58/10 JMP Q24:3 EOR
%   N7:58/10  T_W3 %
% Rung: 4 %
SOR XIC N7:58/11 JMP Q24:4 EOR
%   N7:58/11  T_W4 %
% Rung: 5 %
SOR XIC N7:58/12 JMP Q24:5 EOR
%   N7:58/12  T_W5 %
% Rung: 6 %
SOR XIC N7:58/13 JMP Q24:6 EOR
%   N7:58/13  T_W6 %
% Rung: 7 %
SOR XIC N7:58/14 JMP Q24:7 EOR
%   N7:58/14  T_W7 %
% Rung: 8 %
SOR XIC N7:58/15 JMP Q24:8 EOR
%   N7:58/15  T_W8 %
% Rung: 9 %
SOR LBL Q24:1 OTL N7:58/8 EOR
%   N7:58/8  T_W1 %
% Rung: 10 %
SOR XIO I:2.0/7 JMP Q24:9 EOR
%   I:2.0/7  FO  "Forma otevrena" %

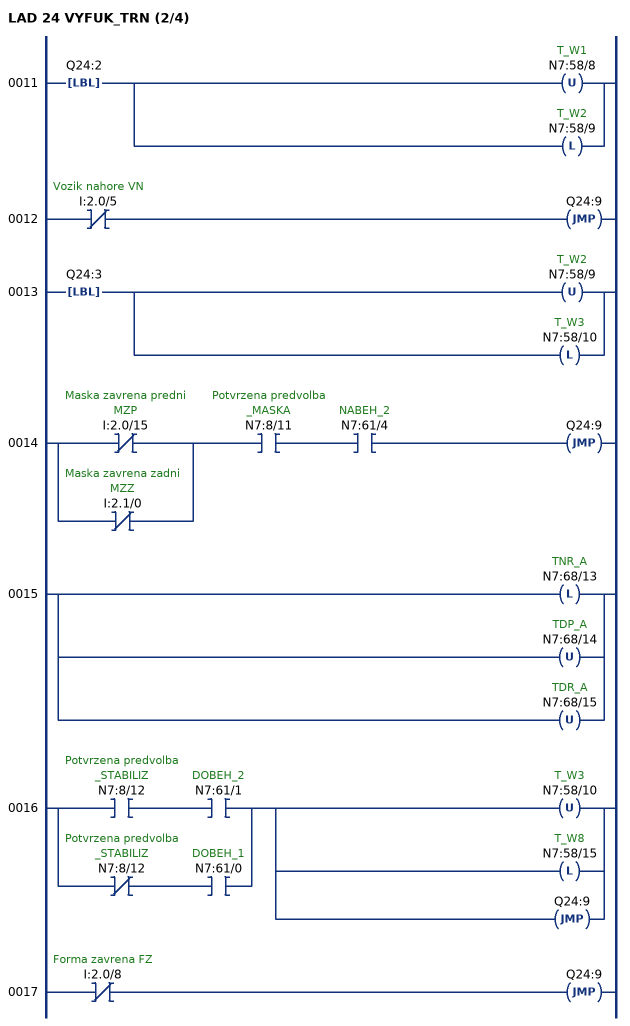
% Rung: 11 %
SOR LBL Q24:2 BST OTU N7:58/8 NXB OTL N7:58/9 BND EOR
%   N7:58/8  T_W1 %
%   N7:58/9  T_W2 %
% Rung: 12 %
SOR XIO I:2.0/5 JMP Q24:9 EOR
%   I:2.0/5  VN  "Vozik nahore" %
% Rung: 13 %
SOR LBL Q24:3 BST OTU N7:58/9 NXB OTL N7:58/10 BND EOR
%   N7:58/9  T_W2 %
%   N7:58/10  T_W3 %
% Rung: 14 %
SOR BST XIO I:2.0/15 NXB XIO I:2.1/0 BND XIC N7:8/11 XIC N7:61/4 JMP Q24:9 EOR
%   I:2.0/15  MZP  "Maska zavrena predni" %
%   I:2.1/0  MZZ  "Maska zavrena zadni" %
%   N7:8/11  _MASKA  "Potvrzena predvolba" %
%   N7:61/4  NABEH_2 %
% Rung: 15 %
SOR BST OTL N7:68/13 NXB BST OTU N7:68/14 NXB OTU N7:68/15 BND BND EOR
%   N7:68/13  TNR_A %
%   N7:68/14  TDP_A %
%   N7:68/15  TDR_A %
% Rung: 16 %
SOR BST XIC N7:8/12 XIC N7:61/1 NXB XIO N7:8/12 XIC N7:61/0 BND BST OTU N7:58/10 NXB OTL N7:58/15 NXB JMP Q24:9 BND EOR
%   N7:8/12  _STABILIZ  "Potvrzena predvolba" %
%   N7:61/1  DOBEH_2 %
%   N7:61/0  DOBEH_1 %
%   N7:58/10  T_W3 %
%   N7:58/15  T_W8 %
% Rung: 17 %
SOR XIO I:2.0/8 JMP Q24:9 EOR
%   I:2.0/8  FZ  "Forma zavrena" %

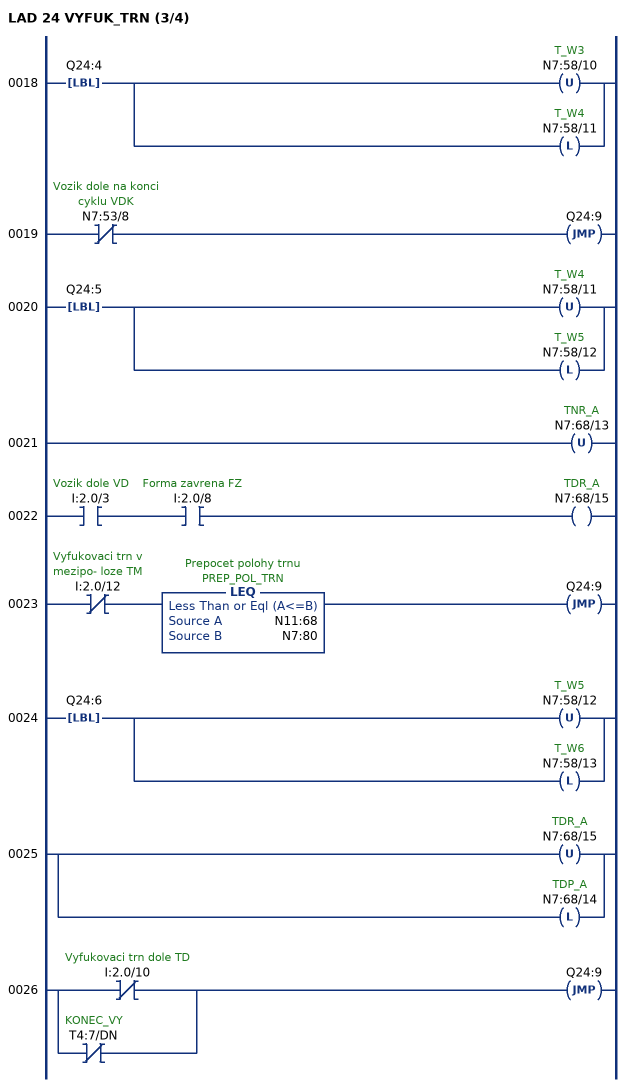
% Rung: 18 %
SOR LBL Q24:4 BST OTU N7:58/10 NXB OTL N7:58/11 BND EOR
%   N7:58/10  T_W3 %
%   N7:58/11  T_W4 %
% Rung: 19 %
SOR XIO N7:53/8 JMP Q24:9 EOR
%   N7:53/8  VDK  "Vozik dole na konci cyklu" %
% Rung: 20 %
SOR LBL Q24:5 BST OTU N7:58/11 NXB OTL N7:58/12 BND EOR
%   N7:58/11  T_W4 %
%   N7:58/12  T_W5 %
% Rung: 21 %
SOR OTU N7:68/13 EOR
%   N7:68/13  TNR_A %
% Rung: 22 %
SOR XIC I:2.0/3 XIC I:2.0/8 OTE N7:68/15 EOR
%   I:2.0/3  VD  "Vozik dole" %
%   I:2.0/8  FZ  "Forma zavrena" %
%   N7:68/15  TDR_A %
% Rung: 23 %
SOR XIO I:2.0/12 LEQ N11:68 N7:80 JMP Q24:9 EOR
%   I:2.0/12  TM  "Vyfukovaci trn v mezipo- loze" %
%   N11:68  PREP_POL_TRN  "Prepocet polohy trnu" %
% Rung: 24 %
SOR LBL Q24:6 BST OTU N7:58/12 NXB OTL N7:58/13 BND EOR
%   N7:58/12  T_W5 %
%   N7:58/13  T_W6 %
% Rung: 25 %
SOR BST OTU N7:68/15 NXB OTL N7:68/14 BND EOR
%   N7:68/15  TDR_A %
%   N7:68/14  TDP_A %
% Rung: 26 %
SOR BST XIO I:2.0/10 NXB XIO T4:7/DN BND JMP Q24:9 EOR
%   I:2.0/10  TD  "Vyfukovaci trn dole" %
%   T4:7/DN  KONEC_VY %

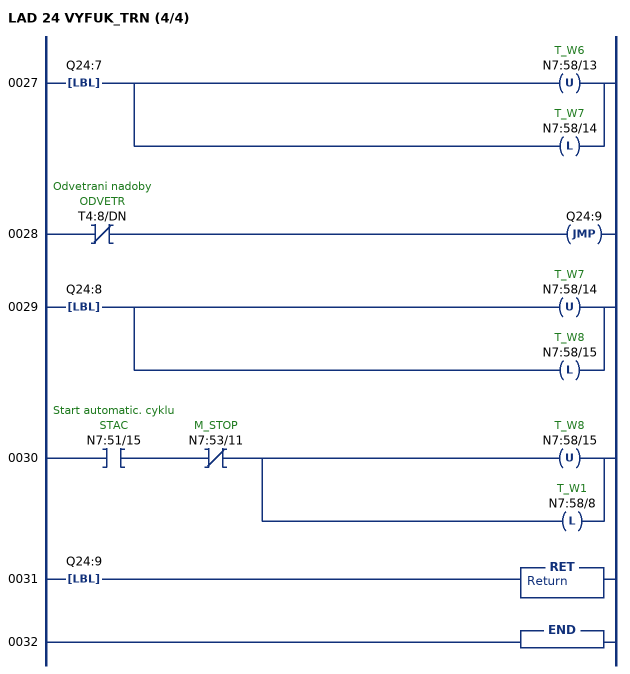
% Rung: 27 %
SOR LBL Q24:7 BST OTU N7:58/13 NXB OTL N7:58/14 BND EOR
%   N7:58/13  T_W6 %
%   N7:58/14  T_W7 %
% Rung: 28 %
SOR XIO T4:8/DN JMP Q24:9 EOR
%   T4:8/DN  ODVETR  "Odvetrani nadoby" %
% Rung: 29 %
SOR LBL Q24:8 BST OTU N7:58/14 NXB OTL N7:58/15 BND EOR
%   N7:58/14  T_W7 %
%   N7:58/15  T_W8 %
% Rung: 30 %
SOR XIC N7:51/15 XIO N7:53/11 BST OTU N7:58/15 NXB OTL N7:58/8 BND EOR
%   N7:51/15  STAC  "Start automatic. cyklu" %
%   N7:53/11  M_STOP %
%   N7:58/15  T_W8 %
%   N7:58/8  T_W1 %
% Rung: 31 %
SOR LBL Q24:9 RET EOR
% Rung: 32 %
SOR END EOR

LADDER 25 "CO2"
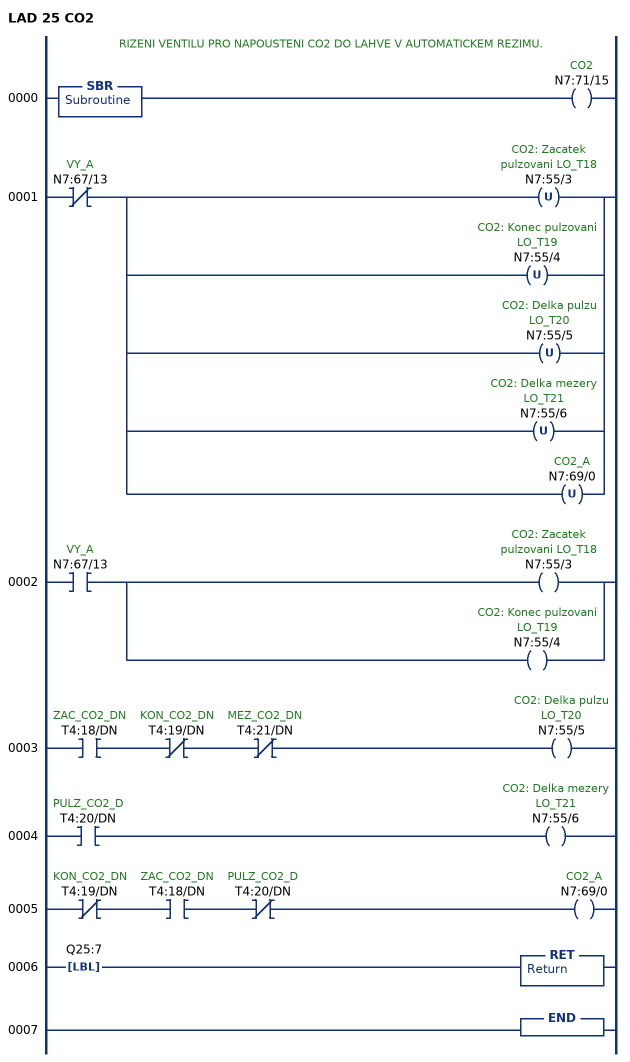
% Rung: 0 %
% RIZENI VENTILU PRO NAPOUSTENI CO2 DO LAHVE V AUTOMATICKEM REZIMU. %
SOR SBR OTE N7:71/15 EOR
%   N7:71/15  CO2 %
% Rung: 1 %
SOR XIO N7:67/13 BST OTU N7:55/3 NXB OTU N7:55/4 NXB OTU N7:55/5 NXB OTU N7:55/6 NXB OTU N7:69/0 BND EOR
%   N7:67/13  VY_A %
%   N7:55/3  LO_T18  "CO2: Zacatek pulzovani" %
%   N7:55/4  LO_T19  "CO2: Konec pulzovani" %
%   N7:55/5  LO_T20  "CO2: Delka pulzu" %
%   N7:55/6  LO_T21  "CO2: Delka mezery" %
%   N7:69/0  CO2_A %
% Rung: 2 %
SOR XIC N7:67/13 BST OTE N7:55/3 NXB OTE N7:55/4 BND EOR
%   N7:67/13  VY_A %
%   N7:55/3  LO_T18  "CO2: Zacatek pulzovani" %
%   N7:55/4  LO_T19  "CO2: Konec pulzovani" %
% Rung: 3 %
SOR XIC T4:18/DN XIO T4:19/DN XIO T4:21/DN OTE N7:55/5 EOR
%   T4:18/DN  ZAC_CO2_DN %
%   T4:19/DN  KON_CO2_DN %
%   T4:21/DN  MEZ_CO2_DN %
%   N7:55/5  LO_T20  "CO2: Delka pulzu" %
% Rung: 4 %
SOR XIC T4:20/DN OTE N7:55/6 EOR
%   T4:20/DN  PULZ_CO2_D %
%   N7:55/6  LO_T21  "CO2: Delka mezery" %
% Rung: 5 %
SOR XIO T4:19/DN XIC T4:18/DN XIO T4:20/DN OTE N7:69/0 EOR
%   T4:19/DN  KON_CO2_DN %
%   T4:18/DN  ZAC_CO2_DN %
%   T4:20/DN  PULZ_CO2_D %
%   N7:69/0  CO2_A %
% Rung: 6 %
SOR LBL Q25:7 RET EOR
% Rung: 7 %
SOR END EOR

LADDER 26 "VYSTUPY"
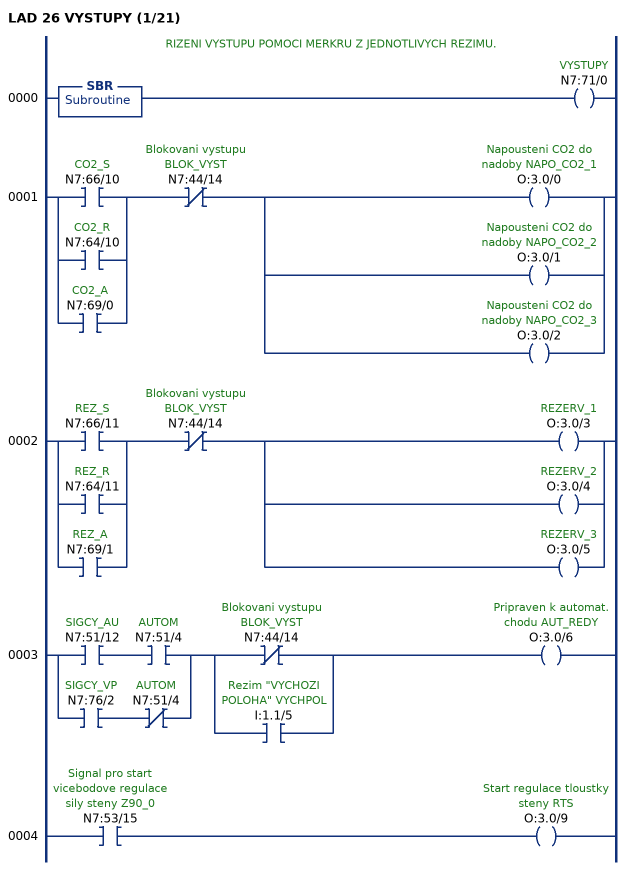
% Rung: 0 %
% RIZENI VYSTUPU POMOCI MERKRU Z JEDNOTLIVYCH REZIMU. %
SOR SBR OTE N7:71/0 EOR
%   N7:71/0  VYSTUPY %
% Rung: 1 %
SOR BST XIC N7:66/10 NXB XIC N7:64/10 NXB XIC N7:69/0 BND XIO N7:44/14 BST OTE O:3.0/0 NXB OTE O:3.0/1 NXB OTE O:3.0/2 BND EOR
%   N7:66/10  CO2_S %
%   N7:64/10  CO2_R %
%   N7:69/0  CO2_A %
%   N7:44/14  BLOK_VYST  "Blokovani vystupu" %
%   O:3.0/0  NAPO_CO2_1  "Napousteni CO2 do nadoby" %
%   O:3.0/1  NAPO_CO2_2  "Napousteni CO2 do nadoby" %
%   O:3.0/2  NAPO_CO2_3  "Napousteni CO2 do nadoby" %
% Rung: 2 %
SOR BST XIC N7:66/11 NXB XIC N7:64/11 NXB XIC N7:69/1 BND XIO N7:44/14 BST OTE O:3.0/3 NXB OTE O:3.0/4 NXB OTE O:3.0/5 BND EOR
%   N7:66/11  REZ_S %
%   N7:64/11  REZ_R %
%   N7:69/1  REZ_A %
%   N7:44/14  BLOK_VYST  "Blokovani vystupu" %
%   O:3.0/3  REZERV_1 %
%   O:3.0/4  REZERV_2 %
%   O:3.0/5  REZERV_3 %
% Rung: 3 %
SOR BST XIC N7:51/12 XIC N7:51/4 NXB XIC N7:76/2 XIO N7:51/4 BND BST XIO N7:44/14 NXB XIC I:1.1/5 BND OTE O:3.0/6 EOR
%   N7:51/12  SIGCY_AU %
%   N7:51/4  AUTOM %
%   N7:76/2  SIGCY_VP %
%   N7:44/14  BLOK_VYST  "Blokovani vystupu" %
%   I:1.1/5  VYCHPOL  "Rezim "VYCHOZI POLOHA"" %
%   O:3.0/6  AUT_REDY  "Pripraven k automat. chodu" %
% Rung: 4 %
SOR XIC N7:53/15 OTE O:3.0/9 EOR
%   N7:53/15  Z90_0  "Signal pro start vicebodove regulace sily steny" %
%   O:3.0/9  RTS  "Start regulace tloustky steny" %

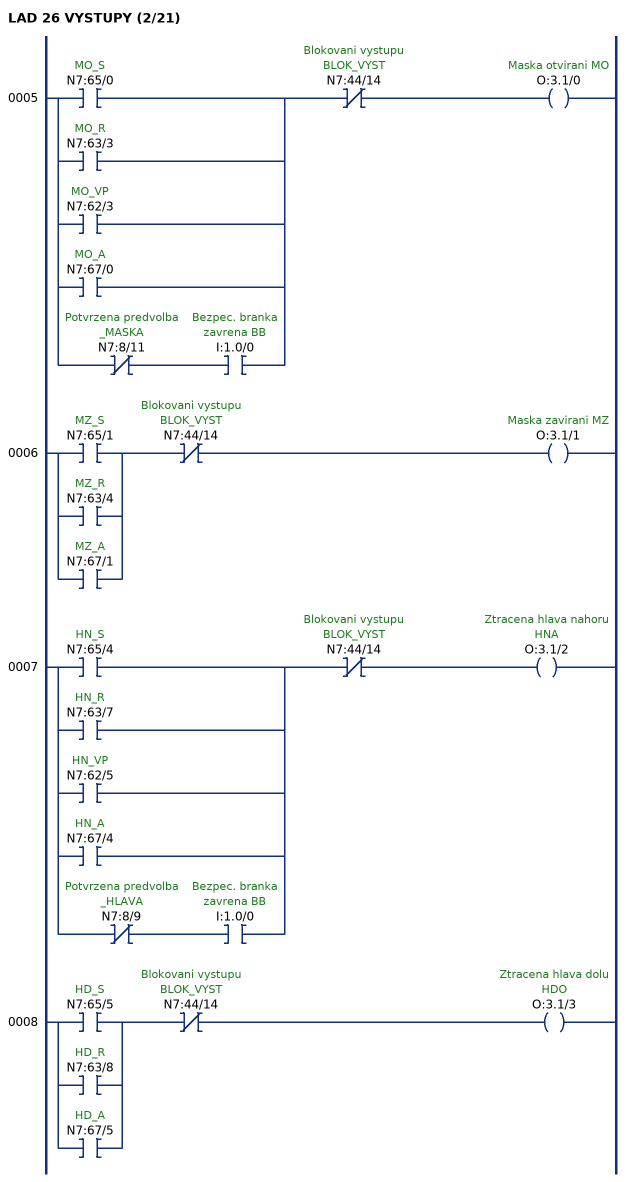
% Rung: 5 %
SOR BST XIC N7:65/0 NXB XIC N7:63/3 NXB XIC N7:62/3 NXB XIC N7:67/0 NXB XIO N7:8/11 XIC I:1.0/0 BND XIO N7:44/14 OTE O:3.1/0 EOR
%   N7:65/0  MO_S %
%   N7:63/3  MO_R %
%   N7:62/3  MO_VP %
%   N7:67/0  MO_A %
%   N7:8/11  _MASKA  "Potvrzena predvolba" %
%   I:1.0/0  BB  "Bezpec. branka zavrena" %
%   N7:44/14  BLOK_VYST  "Blokovani vystupu" %
%   O:3.1/0  MO  "Maska otvirani" %
% Rung: 6 %
SOR BST XIC N7:65/1 NXB XIC N7:63/4 NXB XIC N7:67/1 BND XIO N7:44/14 OTE O:3.1/1 EOR
%   N7:65/1  MZ_S %
%   N7:63/4  MZ_R %
%   N7:67/1  MZ_A %
%   N7:44/14  BLOK_VYST  "Blokovani vystupu" %
%   O:3.1/1  MZ  "Maska zavirani" %
% Rung: 7 %
SOR BST XIC N7:65/4 NXB XIC N7:63/7 NXB XIC N7:62/5 NXB XIC N7:67/4 NXB XIO N7:8/9 XIC I:1.0/0 BND XIO N7:44/14 OTE O:3.1/2 EOR
%   N7:65/4  HN_S %
%   N7:63/7  HN_R %
%   N7:62/5  HN_VP %
%   N7:67/4  HN_A %
%   N7:8/9  _HLAVA  "Potvrzena predvolba" %
%   I:1.0/0  BB  "Bezpec. branka zavrena" %
%   N7:44/14  BLOK_VYST  "Blokovani vystupu" %
%   O:3.1/2  HNA  "Ztracena hlava nahoru" %
% Rung: 8 %
SOR BST XIC N7:65/5 NXB XIC N7:63/8 NXB XIC N7:67/5 BND XIO N7:44/14 OTE O:3.1/3 EOR
%   N7:65/5  HD_S %
%   N7:63/8  HD_R %
%   N7:67/5  HD_A %
%   N7:44/14  BLOK_VYST  "Blokovani vystupu" %
%   O:3.1/3  HDO  "Ztracena hlava dolu" %

